Staubli VAL3: buildList.pgx

program buildList()
  local num i
  local bool l_bFound
  local num l_nCount
  local num l_nSize
  local string l_sEmpty
  local string l_sEvent
begin
  // INIT the list
  l_sEmpty=""
  call use:stringCopy(l_sEmpty,sList)
  // Build the list
  call home:getBoxSize(save:nBoxType,l_nSize)
  for i=0 to l_nSize-1
    call set:getEvent(l_sEvent,i,save:nBoxType)
    if l_sEvent!=""
      //
      // use the filter ?
      //
      // check if the bProcessList filter is active
      //
      l_bFound=true
      // update the selected item
      if l_sEvent==sEvent
        nSelected=l_nCount
      endIf
      // add
      if l_bFound
        call listAdd(l_sEvent)
        l_nCount=l_nCount+1
      endIf
    endIf
  endFor
  // update
  use:bUseRefresh=true
end
